{attribute 'qualified_only'}
VAR_GLOBAL
END_VAR

(* stored: Version 1.1.0.1, ProductVersion 3.1.4022.7
   GVL GVL_02_Parameter_Step_Motor_Other: Id {571e8aa8-3118-4aba-b296-e589e8661db9} *)
